(* CODESYS project Dry-Martini.project

Project tree, tasks and I/O mapping:
  Device : CODESYS Control Win V3, 3S - Smart Software Solutions GmbH, order no. 305021, version 3.5.6.10
    application Application
      libraries: Standard, * (System)
      task MainTask (cyclic, interval t#20ms, priority 1) calls Main, Desl_EMG, Escoamento_EMG
      task Modo_Area (cyclic, interval t#20ms, priority 1) calls Auto_A1, Auto_A2, Manual_A1, Manual_A2
      task Temperatura (cyclic, interval t#500ms, priority 2) calls Temp_Prod
      task Vazao_Gin (cyclic, interval t#50ms, priority 2) calls Vaz_Gin
      task Vazao_Vermounth (cyclic, interval t#50ms, priority 2) calls Vaz_Verm
      task Vazao_Refrigerante (cyclic, interval t#5ms, priority 2) calls Vaz_Refri_E, Vaz_Refri_S
      task Vazao_DryMartini (cyclic, interval t#50ms, priority 1) calls Vaz_DryMartini
      task Vazao_Bico (cyclic, interval t#50ms, priority 1) calls Vaz_Bico
      global variables GLOBAL
      global variables GLOBAL_A1
      program Auto_A1 [SFC]: Nivel_Refri, Tot_Gin, Tot_Verm, Agitador_A, Valv_Ref_A, Valv_Ref_D, Temp_Refri, Agitador_D, Valv_Transicao, Bomba, Nivel_RM01, Re_Ini, Desab_Escoa
      program Main [SFC]: Automatico_OP, Manual_OP
      program Vaz_Gin [ST]
      program Vaz_Verm [ST]
      program Vaz_Refri_E [ST]
      program Temp_Prod [ST]
      program Vaz_DryMartini [ST]
      global variables GLOBAL_A2
      program Vaz_Refri_S [ST]
      program Auto_A2 [SFC]: Nivel_10, Nivel_TP01_B, Motor, S_Proxi, Re_Ini, Tot_Dry, Ini_Count, T_Tonel, Nivel_95
      program Vaz_Bico [ST]
      program Desl_EMG [SFC]: Imediato, Em_3_S, Em_5_S, Reseta_V_EMG
      program Manual_A1 [SFC]
      program Manual_A2 [SFC]
      program Escoamento_EMG [SFC]: Escoamento, Re_Ini
*)

// Device/Application/GLOBAL
VAR_GLOBAL
	
// TOTALIZADORES
	FQ04:REAL:=0;  				// Quanto de Dry-Martine foi produzido ao todo

// EMERGENCIA
	EMG:BOOL:=FALSE; 			// Botao de EMERGENCIA
	Acao1:BOOL:=FALSE; 			// Primeira ACAO a ser realizada pela EMERGENCIA
	Acao2:BOOL:=FALSE; 			// Segunda ACAO a ser realizada apos 3S pela EMERGENCIA
	Acao3:BOOL:=FALSE; 			// Segunda ACAO a ser realizada apos 5S pela EMERGENCIA
	Aux_Esc_EMG:BOOL:=FALSE; 	// Habilita o ESCOAMENTO DE EMERGENCIA que esvazia o tanque
	Esc_EMG:BOOL:=FALSE; 		// Aciona o ESCOAMENTO DE EMERGENCIA que esvazia o tanque

// VARIAVEIS GLOBAIS QUE NÃO SÃO DESCRITAS EM NENHUMA AREA
// ------------------------------------------------------- //
	// ACIONA
	Liga:BOOL;					// Liga o PROCESSO
	Modo:BOOL;					// SELECIONA o modo de OPERAÇÃO do processo
		
// ------------------------------------------------------- //	

END_VAR

// Device/Application/GLOBAL_A1
VAR_GLOBAL

// VALVULAS AREA 01
	FV101	:BOOL; // Reservtorio GIN
	FV102	:BOOL; // Reservtorio VERMOUNTH
	FV103	:BOOL; // Reservtorio LIQUIDO REFRIGERANTE (ENTRADA)
	FV104	:BOOL; // Saida MOTOR BA-101
	FV105	:BOOL; // Transisção AREA01 a AREA02
	FV106	:BOOL; // DRENO
	FV107	:BOOL; // Reservtorio LIQUIDO REFRIGERANTE (SAIDA)

// SENSORES DE NIVEL (JAQUETA)
	LSL102	:BOOL; // Sensor de Nivel Baixo (MINIMO DE DETECÇÃO 0.005 LITROS OU 5mL(TRUE))
	LSH102	:BOOL; // Sensor de Nivel Alto
	
// SENSORES DE NIVEL (RESERVATORIO)
	LSL101	:BOOL; // Sensor de Nivel Baixo
	LSH101	:BOOL; // Sensor de Nivel até a jaqueta
	LT101	:REAL;  // Sensor de Nivel Total

// SENSORES DE TEMPERATURA
	TSL101	:BOOL; // Sensor de Temperatura
	
// MOTORES
	BA101	:BOOL; // Motor de fluido AREA01 a AREA02
	M101	:BOOL; // Motor do Agitador
	
// TOTALIZADORES
	FQ101:REAL:=0; // GIN (Litros)
	FQ102:REAL:=0; // VERMOUNTH (Litros)
	FQ103:REAL:=0; // DRYMARTINI (Litros)
	
// FALHAS
	Falha_N_RM01:BOOL:=FALSE;


// ----------------- VARIAVEIS DE PROCESSO A1 (NÃO ESTÃO NO ESCOPO) ---------------------//
	
	// ACIONAMENTO
	Liga_Auto:BOOL; // Variavel de acionamento AUTOMATICO
		
	// NIVEL
	Nivel_Jaqueta:REAL; // Nivel do Liquido Refrigerante na jaqueta
	Reserv_Vazio:BOOL; // Verifica se o tanque está TOTALMENTE vazio
	
	// TEMPERATURA
	Temp_Produto:REAL := 25.0; // Temperatura Inicial dos Componentes-Base (GIN e VERMOUNTH)
	Simul_Decai:BOOL; // Habilita a SIMULAÇAO de DECAIMENTO da temperatura
	
	
END_VAR

// Device/Application/GLOBAL_A2
VAR_GLOBAL
	
// VALVULAS AREA 02
	FV201	:BOOL; // Saida Tanque de Produto
		
// SENSORES DE NIVEL (TANQUE DE PRODUTO)
	LSL201	:BOOL; // Sensor de Nivel Baixo
	LSH201	:BOOL; // Sensor de Nivel Alto
	LSHH201	:BOOL; // Sensor de Nivel Alto-Alto
	LT201	:REAL;  // Sensor de Nivel Total
	
// TOTALIZADORES
	FQ201:REAL:=0; // TONEL (Litros)

// SENSORES DIVERSOS
	ZY201:BOOL; // Sensor de Proximadade BICO
	ZY202:BOOL; // Sensor Capacitivo CONTADOR
	
// MOTORES
	M201:BOOL; // Motor ESTEIRA
		


// ----------------- VARIAVEIS DE PROCESSO A2 (NÃO ESTÃO NO ESCOPO)----------------------//
	
	// ACIONAMENTO
	Inicia_TP:BOOL; // Habita a Segunda Area 02
	
	// FALHA
	Falha_Q_Tonel:BOOL; // Habilita o transporte vazio (PARA TESTE)
	
	// MENSAGENS (OUTRAS)
	Transp_Vazio:BOOL; // Mensagem TRANSPORTE VAZIO
	
	
END_VAR

// Device/Application/Main
PROGRAM Main
VAR
END_VAR

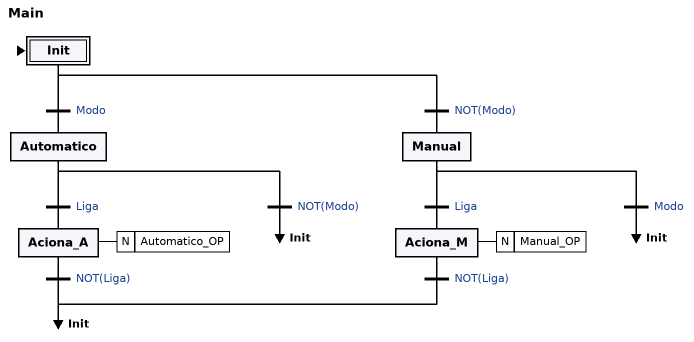
INITIAL_STEP Init:
END_STEP
TRANSITION FROM Init TO Automatico
    := Modo;
END_TRANSITION
STEP Automatico:
END_STEP
TRANSITION FROM Automatico TO Aciona_A
    := Liga;
END_TRANSITION
TRANSITION FROM Automatico TO Init
    := NOT(Modo);
END_TRANSITION
STEP Aciona_A:
    Automatico_OP(N);
END_STEP
TRANSITION FROM Aciona_A TO Init
    := NOT(Liga);
END_TRANSITION
TRANSITION FROM Init TO Manual
    := NOT(Modo);
END_TRANSITION
STEP Manual:
END_STEP
TRANSITION FROM Manual TO Aciona_M
    := Liga;
END_TRANSITION
TRANSITION FROM Manual TO Init
    := Modo;
END_TRANSITION
STEP Aciona_M:
    Manual_OP(N);
END_STEP
TRANSITION FROM Aciona_M TO Init
    := NOT(Liga);
END_TRANSITION

ACTION Automatico_OP:
Liga_Auto := Aciona_A.x;
END_ACTION

ACTION Manual_OP:

END_ACTION

END_PROGRAM

// Device/Application/Desl_EMG
PROGRAM Desl_EMG
VAR
END_VAR

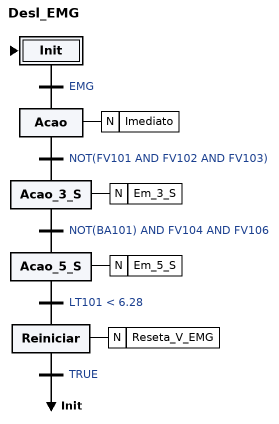
INITIAL_STEP Init:
END_STEP
TRANSITION FROM Init TO Acao
    := EMG;
END_TRANSITION
STEP Acao:
    Imediato(N);
END_STEP
TRANSITION FROM Acao TO Acao_3_S
    := NOT(FV101 AND FV102 AND FV103);
END_TRANSITION
STEP Acao_3_S:
    Em_3_S(N);
END_STEP
TRANSITION FROM Acao_3_S TO Acao_5_S
    := NOT(BA101) AND FV104 AND FV106;
END_TRANSITION
STEP Acao_5_S:
    Em_5_S(N);
END_STEP
TRANSITION FROM Acao_5_S TO Reiniciar
    := LT101 < 6.28;
END_TRANSITION
STEP Reiniciar:
    Reseta_V_EMG(N);
END_STEP
TRANSITION FROM Reiniciar TO Init
    := TRUE;
END_TRANSITION

ACTION Imediato:
// Deligar Valvulas GIN, VERMOUNTH e LIQUIDO REFRIGERANTE
IF(Acao.x)THEN
	Acao1 := Acao.x;
	FV101 := FALSE;
	FV102 := FALSE;
	FV103 := FALSE;
END_IF
END_ACTION

ACTION Em_3_S:
// Apos 3S = Deligar o Motor BOMBA e Ligar as Valvulas FV-104 e FV-106
IF(Acao_3_S.x)THEN
	Acao2 := Acao_3_S.x;
	BA101 := FALSE;
	FV104 := TRUE;
	FV106 := TRUE;
END_IF
END_ACTION

ACTION Em_5_S:
// Apos 5S = Ligar o Motor BOMBA ate LSL-101 (IDEIA DE 10%)
IF(Acao_5_S.x AND LT101 < 6.28)THEN
	Acao3 := Acao_5_S.x;
	BA101 := TRUE;
END_IF
END_ACTION

ACTION Reseta_V_EMG:
BA101 := FALSE;
FV104 := FALSE;
FV106 := FALSE;
Aux_Esc_EMG := TRUE;
Liga := FALSE;
END_ACTION

END_PROGRAM

// Device/Application/Escoamento_EMG
PROGRAM Escoamento_EMG
VAR
END_VAR

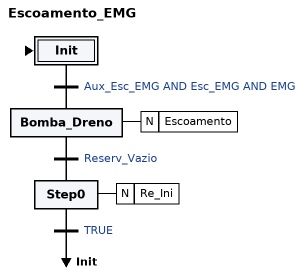
INITIAL_STEP Init:
END_STEP
TRANSITION FROM Init TO Bomba_Dreno
    := Aux_Esc_EMG AND Esc_EMG AND EMG;
END_TRANSITION
STEP Bomba_Dreno:
    Escoamento(N);
END_STEP
TRANSITION FROM Bomba_Dreno TO Step0
    := Reserv_Vazio;
END_TRANSITION
STEP Step0:
    Re_Ini(N);
END_STEP
TRANSITION FROM Step0 TO Init
    := TRUE;
END_TRANSITION

ACTION Escoamento:
// Aciona o DRENO
FV104 := TRUE;
BA101 := TRUE;
FV106 := TRUE;
END_ACTION

ACTION Re_Ini:
// Desaciona o DRENO
FV104 := FALSE;
BA101 := FALSE;
FV106 := FALSE;
END_ACTION

END_PROGRAM

// Device/Application/Auto_A1
PROGRAM Auto_A1
VAR
	TON1: TON; // TEMPORIZADOR
	AUX01: BOOL;
END_VAR
VAR // added by the converter: edge detectors and wires of the graphical bodies
    _w1 : BOOL;
END_VAR

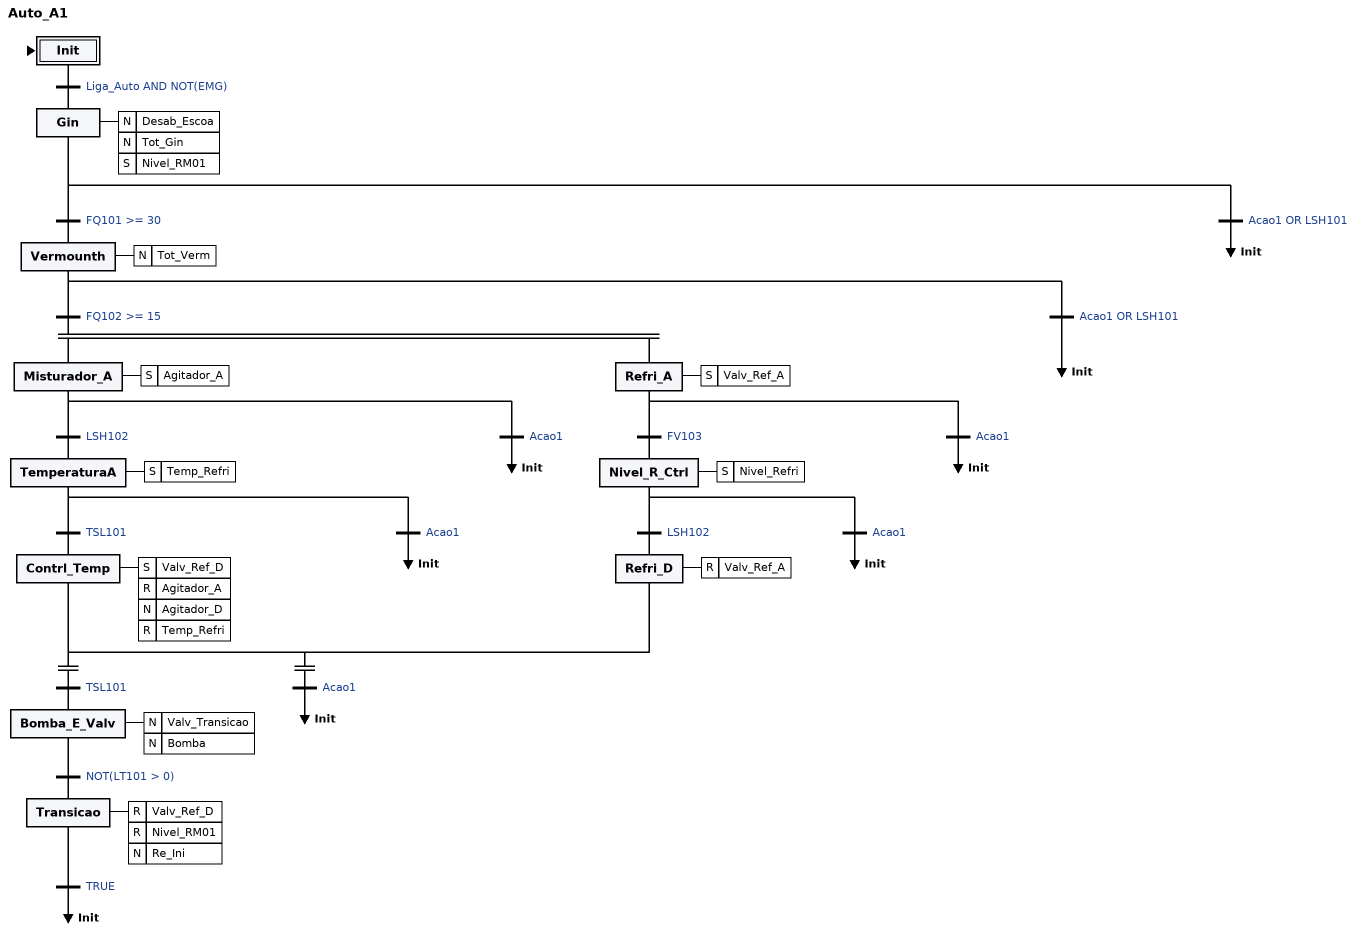
INITIAL_STEP Init:
END_STEP
TRANSITION FROM Init TO Gin
    := Liga_Auto AND NOT(EMG);
END_TRANSITION
STEP Gin:
    Desab_Escoa(N);
    Tot_Gin(N);
    Nivel_RM01(S);
END_STEP
TRANSITION FROM Gin TO Vermounth
    := FQ101 >= 30;
END_TRANSITION
TRANSITION FROM Gin TO Init
    := Acao1 OR LSH101;
END_TRANSITION
STEP Vermounth:
    Tot_Verm(N);
END_STEP
TRANSITION FROM Vermounth TO (Misturador_A, Refri_A)
    := FQ102 >= 15;
END_TRANSITION
TRANSITION FROM Vermounth TO Init
    := Acao1 OR LSH101;
END_TRANSITION
STEP Misturador_A:
    Agitador_A(S);
END_STEP
TRANSITION FROM Misturador_A TO TemperaturaA
    := LSH102;
END_TRANSITION
TRANSITION FROM Misturador_A TO Init
    := Acao1;
END_TRANSITION
STEP TemperaturaA:
    Temp_Refri(S);
END_STEP
TRANSITION FROM TemperaturaA TO Contrl_Temp
    := TSL101;
END_TRANSITION
TRANSITION FROM TemperaturaA TO Init
    := Acao1;
END_TRANSITION
STEP Contrl_Temp:
    Valv_Ref_D(S);
    Agitador_A(R);
    Agitador_D(N);
    Temp_Refri(R);
END_STEP
STEP Refri_A:
    Valv_Ref_A(S);
END_STEP
TRANSITION FROM Refri_A TO Nivel_R_Ctrl
    := FV103;
END_TRANSITION
TRANSITION FROM Refri_A TO Init
    := Acao1;
END_TRANSITION
STEP Nivel_R_Ctrl:
    Nivel_Refri(S);
END_STEP
TRANSITION FROM Nivel_R_Ctrl TO Refri_D
    := LSH102;
END_TRANSITION
TRANSITION FROM Nivel_R_Ctrl TO Init
    := Acao1;
END_TRANSITION
STEP Refri_D:
    Valv_Ref_A(R);
END_STEP
TRANSITION FROM (Contrl_Temp, Refri_D) TO Bomba_E_Valv
    := TSL101;
END_TRANSITION
TRANSITION FROM (Contrl_Temp, Refri_D) TO Init
    := Acao1;
END_TRANSITION
STEP Bomba_E_Valv:
    Valv_Transicao(N);
    Bomba(N);
END_STEP
TRANSITION FROM Bomba_E_Valv TO Transicao
    := NOT(LT101 > 0);
END_TRANSITION
STEP Transicao:
    Valv_Ref_D(R);
    Nivel_RM01(R);
    Re_Ini(N);
END_STEP
TRANSITION FROM Transicao TO Init
    := TRUE;
END_TRANSITION
// branch label No1

ACTION Nivel_Refri:
// NIVEL BAIXO JAQUETA
IF(Nivel_Jaqueta >= 0.5) THEN
	LSL102 := TRUE;
ELSE
	LSL102 := FALSE;
END_IF

// NIVEL ALTO JAQUETA
IF(Nivel_Jaqueta >= 5.0) THEN
	LSH102 := TRUE;
ELSE
	LSH102 := FALSE;
END_IF
END_ACTION

ACTION Tot_Gin:
// Aciona Valvula de GIN
FV101 := Gin.x;
END_ACTION

ACTION Tot_Verm:
// Aciona Valvula de VERMOUNTH
FV102 := Vermounth.x;
END_ACTION

ACTION Agitador_A:
// Aciona Motor do MISTURADOR
M101 := TRUE;

// ALTO (Para NOVAS bateladas)
//IF(LT101 >= 50)THEN
//	LSH101 := TRUE;
//	Liga_Auto:=FALSE;
//	Falha_N_RM01:=TRUE;
//	Liga:=FALSE;
//ELSE
//	LSH101 := FALSE;
//END_IF
END_ACTION

ACTION Valv_Ref_A:
// Aciona Valvula de ENTRADA de LIQUIDO REFRIGERANTE
FV103 := TRUE AND NOT(LSH102);
END_ACTION

ACTION Valv_Ref_D:
// Aciona Valvula de SAIDA de LIQUIDO REFRIGERANTE
IF(LSL102)THEN
	FV107 := TRUE;
ELSE
	FV107 := FALSE;
END_IF
END_ACTION

ACTION Temp_Refri:
// A TEMPERATURA SERÁ ALTERADA QUANTO FOR ADICIONADO O LIQ. REFRIGERANTE
Simul_Decai:= LSH102 AND NOT(TSL101);
END_ACTION

ACTION Agitador_D:
// Desativa o Motor do MISTURADOR
M101:=FALSE;
END_ACTION

ACTION Valv_Transicao:
// Acionamento das Valvulas de TRANSMISSAO de DRY-MARTINI
IF(Bomba_E_Valv.x AND NOT(Reserv_Vazio))THEN
	FV104 := TRUE;
	FV105 := TRUE;
ELSE
	FV104 := FALSE;
	FV105 := FALSE;
END_IF
END_ACTION

ACTION Bomba:
// ACIONA BOMBA
IF(Bomba_E_Valv.x AND NOT(Reserv_Vazio))THEN
	BA101 := TRUE;
ELSE
	BA101 := FALSE;
END_IF
END_ACTION

ACTION Nivel_RM01:
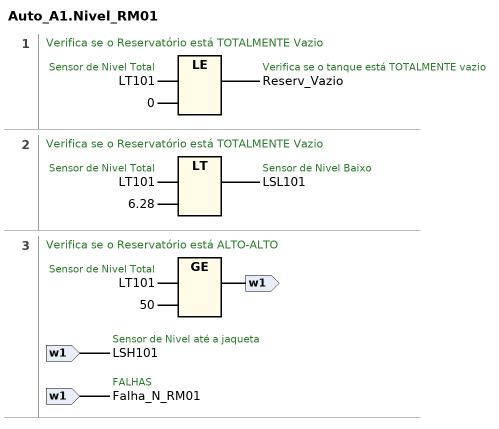
// NETWORK 1
// Verifica se o Reservatório está TOTALMENTE Vazio
//   LT101: Sensor de Nivel Total
//   Reserv_Vazio: Verifica se o tanque está TOTALMENTE vazio
Reserv_Vazio := LT101 <= 0;

// NETWORK 2
// Verifica se o Reservatório está TOTALMENTE Vazio
//   LT101: Sensor de Nivel Total
//   LSL101: Sensor de Nivel Baixo
LSL101 := LT101 < 6.28;

// NETWORK 3
// Verifica se o Reservatório está ALTO-ALTO
//   LT101: Sensor de Nivel Total
//   LSH101: Sensor de Nivel até a jaqueta
//   Falha_N_RM01: FALHAS
_w1 := LT101 >= 50;
LSH101 := _w1;
Falha_N_RM01 := _w1;
END_ACTION

ACTION Re_Ini:
// TOTALIZADOR GERAL E ZERAR O TOTALIZADOR DRY-MARTINI
FQ103:=0;
Temp_Produto := 25.0;
FQ101 := 0;
FQ102 := 0;
FQ103 := 0;
Inicia_TP := TRUE;
END_ACTION

ACTION Desab_Escoa:
Aux_Esc_EMG := FALSE;
END_ACTION

END_PROGRAM

// Device/Application/Auto_A2
PROGRAM Auto_A2
VAR
	TON1:TON; // TEMPORIZADOR DO SENSOR
	Deteccao:BOOL;
END_VAR

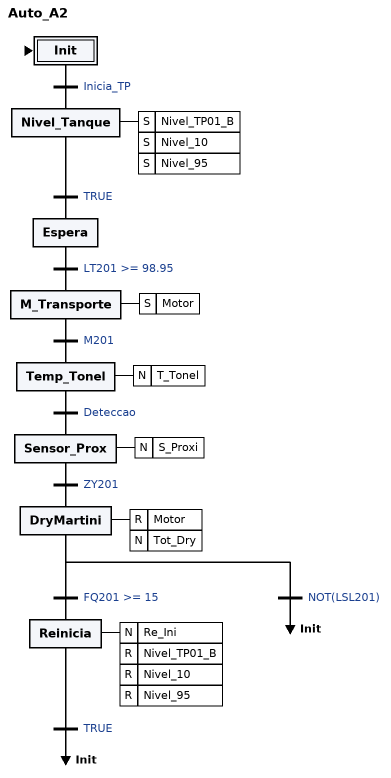
INITIAL_STEP Init:
END_STEP
TRANSITION FROM Init TO Nivel_Tanque
    := Inicia_TP;
END_TRANSITION
STEP Nivel_Tanque:
    Nivel_TP01_B(S);
    Nivel_10(S);
    Nivel_95(S);
END_STEP
TRANSITION FROM Nivel_Tanque TO Espera
    := TRUE;
END_TRANSITION
STEP Espera:
END_STEP
TRANSITION FROM Espera TO M_Transporte
    := LT201 >= 98.95;
END_TRANSITION
STEP M_Transporte:
    Motor(S);
END_STEP
TRANSITION FROM M_Transporte TO Temp_Tonel
    := M201;
END_TRANSITION
STEP Temp_Tonel:
    T_Tonel(N);
END_STEP
TRANSITION FROM Temp_Tonel TO Sensor_Prox
    := Deteccao;
END_TRANSITION
STEP Sensor_Prox:
    S_Proxi(N);
END_STEP
TRANSITION FROM Sensor_Prox TO DryMartini
    := ZY201;
END_TRANSITION
STEP DryMartini:
    Motor(R);
    Tot_Dry(N);
END_STEP
TRANSITION FROM DryMartini TO Reinicia
    := FQ201 >= 15;
END_TRANSITION
TRANSITION FROM DryMartini TO Init
    := NOT(LSL201);
END_TRANSITION
STEP Reinicia:
    Re_Ini(N);
    Nivel_TP01_B(R);
    Nivel_10(R);
    Nivel_95(R);
END_STEP
TRANSITION FROM Reinicia TO Init
    := TRUE;
END_TRANSITION

ACTION Nivel_10:
// AÇÕES de NIVEL 10%
IF(NOT(LSL201))THEN
	FV201:= FALSE;
	M201:= FALSE;
END_IF
END_ACTION

ACTION Nivel_TP01_B:
// SENSORES BOOLEANOS

// SENSOR BAIXO
IF(LT201 >= 19.79)THEN
	LSL201 := TRUE;
ELSE
	LSL201 := FALSE;
END_IF

// SENSOR ALTO
IF(LT201 >= 168.215)THEN
	LSH201 := TRUE;
ELSE
	LSH201 := FALSE;
END_IF

// SENSOR ALTO-ALTO
IF(LT201 >= 188.005)THEN
	LSHH201 := TRUE;
ELSE
	LSHH201 := FALSE;
END_IF
END_ACTION

ACTION Motor:
// Aciona Motor da ESTEIRA
M201 := TRUE AND NOT(ZY201);
END_ACTION

ACTION S_Proxi:
// Sensor DETECTA
ZY201:=TRUE;
END_ACTION

ACTION Re_Ini:
// RESETA variaveis para NOVO Ciclo
FV201 := FALSE;
FQ201 := 0;
ZY201 := FALSE;
END_ACTION

ACTION Tot_Dry:
// Aciona Valvula de DRY-MARTINI
IF(DryMartini.x)THEN
	FV201 := TRUE;
ELSE
	FV201 := FALSE;
END_IF
END_ACTION

ACTION Ini_Count:

END_ACTION

ACTION T_Tonel:
// TEMPORIZADOR TONEL
IF((Temp_Tonel.t >= T#5S AND Temp_Tonel.t < T#15S) AND NOT(Falha_Q_Tonel))THEN // TEM TONEL
	Deteccao		:=TRUE;
	Transp_Vazio	:=FALSE;
ELSIF((Temp_Tonel.t >= T#15S ) AND Falha_Q_Tonel)THEN // NAO TEM TONEL
	Deteccao		:=FALSE;
	Transp_Vazio	:=TRUE;
ELSE												 // EM ESPERA
	Deteccao		:=FALSE;
END_IF
END_ACTION

ACTION Nivel_95:
// AÇÕES de NIVEL 95%
IF(LSHH201)THEN
	FV104:= FALSE;
	FV105:= FALSE;
	BA101:= FALSE;
END_IF
END_ACTION

END_PROGRAM

// Device/Application/Manual_A1
PROGRAM Manual_A1
VAR
END_VAR

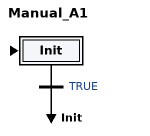
INITIAL_STEP Init:
END_STEP
TRANSITION FROM Init TO Init
    := TRUE;
END_TRANSITION

END_PROGRAM

// Device/Application/Manual_A2
PROGRAM Manual_A2
VAR
END_VAR

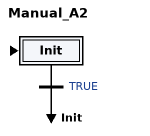
INITIAL_STEP Init:
END_STEP
TRANSITION FROM Init TO Init
    := TRUE;
END_TRANSITION

END_PROGRAM

// Device/Application/Temp_Prod
PROGRAM Temp_Prod
VAR
END_VAR

// SIMULA decaimento de TEMPERATURA
IF(LSH102)THEN // TEM LIQUIDO REFRIGERANTE
	Temp_Produto := Temp_Produto - 0.5;
END_IF

IF(Temp_Produto > 1)THEN
	TSL101 := FALSE;
ELSE
	TSL101 := TRUE;
END_IF

END_PROGRAM

// Device/Application/Vaz_Gin
PROGRAM Vaz_Gin
VAR
END_VAR

// SIMULA vazao do GIN
IF(FV101)THEN
	FQ101 := FQ101 + 0.3;
	LT101 := LT101 + 0.3;
END_IF

END_PROGRAM

// Device/Application/Vaz_Verm
PROGRAM Vaz_Verm
VAR
END_VAR

// SIMULA vazao do VERMOUNTH
IF(FV102)THEN
	FQ102 := FQ102 + 0.25;
	LT101 := LT101 + 0.25;
END_IF

END_PROGRAM

// Device/Application/Vaz_Refri_E
PROGRAM Vaz_Refri_E
VAR
END_VAR

// SIMULA vazao de entrada do LIQUIDO REFRIGERANTE
// ENTRADA
IF(FV103)THEN
	Nivel_Jaqueta := Nivel_Jaqueta + 0.025;
END_IF

END_PROGRAM

// Device/Application/Vaz_Refri_S
PROGRAM Vaz_Refri_S
VAR
END_VAR

// SIMULA vazao de saida do LIQUIDO REFRIGERANTE
// SAIDA
IF(FV107)THEN
	Nivel_Jaqueta := Nivel_Jaqueta - 0.025;
END_IF

END_PROGRAM

// Device/Application/Vaz_DryMartini
PROGRAM Vaz_DryMartini
VAR

END_VAR

// SIMULA VAZAO DA TRANSMISSAO DE PRODUTO DE RM01 A TP01
IF(FV104 AND BA101 AND FV105)THEN
	FQ103 := FQ103 + 0.75;
	LT101 := LT101 - 0.75;
	LT201 := LT201 + 0.75;
END_IF

// SIMULA VAZAO DO DRENO
IF(FV104 AND BA101 AND FV106)THEN
	LT101 := LT101 - 0.75;
END_IF

END_PROGRAM

// Device/Application/Vaz_Bico
PROGRAM Vaz_Bico
VAR
END_VAR

// SIMULA vazao do BICO
IF(FV201)THEN
	FQ201 := FQ201 + 0.15;
	LT201 := LT201 - 0.15;
END_IF

END_PROGRAM
